(* Schneider Machine Expert - Basic project Control banda, file version 2.9.0.0 *)
(* ProjectInformations: Name=New project *)

HARDWARE
  Cpu 0: TM221CE16R
  EthernetConfiguration: NetworkName=M221, IpAllocationMode=FixedAddress, IpAddress=0.0.0.0, SubnetMask=0.0.0.0
  SerialLineConfiguration: Baud=Baud19200, Parity=ParityEven, DataBits=DataBits8, StopBits=StopBits1, PhysicalMedium=PhysicalMediumRs485, TransmissionMode=TransmissionModeModbusRtu, SlaveId=1, Addressing=SlaveAddressing
  MastTask: UsePeriodScanMode=false, PeriodScan=100
  FastTask: Period=255
  CpuBehavior: StartingMode=StartAsPreviousState, AutoSaveRamOnEeprom=true, WatchdogPeriod=250

SYMBOLS  (address, symbol, comment, settings)
  %M0       AT_EXIT
  %M1       START_FIO
  %M2       RESET_FIO
  %M3       STOP_FIO
  %M4       EMERG_FIO
  %M10      ENTRY_CONVEY
  %M11      STOP_BLAE
  %M12      EXIT_CONVEYOR
  %M13      SORTER_1_TURN
  %M14      SORTER_1_BELT
  %M15      SORTER_2_TURN
  %M16      SORTER_2_BELT
  %M17      SORTER_3_TURN
  %M18      SORTER_3_BELT
  %M19      START_LIGHT
  %M21      STOP_LIGHT
  %M30      START_REMOT
  %M31      STOP_REMOTO
  %M32      PAUSE_REM
  %M33      RESET_REMOT
  %M34      EMERG_REMOTA_
  %M41      BLUE_ACTIVE
  %M42      GREEN_ACTIVE
  %M43      METAL_ACTIVE
  %S6       SB_TB1S  "Time base of 1 s generated by an internal clock"
  %TM0        [Preset=3, Base=OneHundredMilliSeconds]
  %TM1        [Preset=22, Base=OneHundredMilliSeconds]
  %TM2        [Preset=40, Base=OneHundredMilliSeconds]
  %TM10       [Type=TP, Preset=10, Base=OneHundredMilliSeconds]
  %TM11       [Type=TP, Preset=10, Base=OneHundredMilliSeconds]
  %TM12       [Type=TP, Preset=10, Base=OneHundredMilliSeconds]

POU New POU
  (* SectionNumber=1 *)

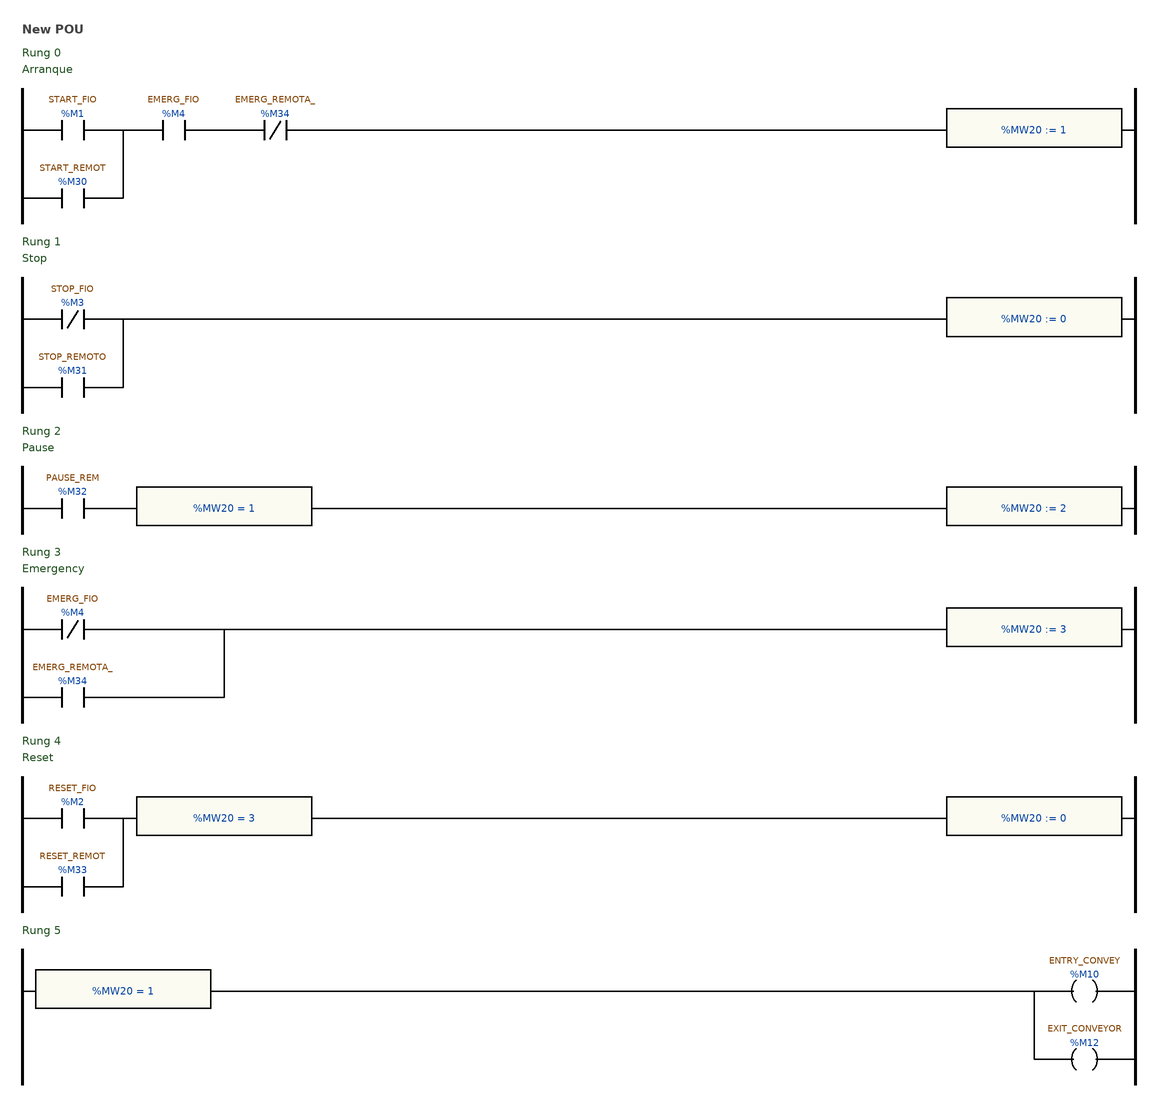

// Rung 0
// Arranque
  LD %M1                  (* START_FIO *)
  OR %M30                 (* START_REMOT *)
  AND %M4                 (* EMERG_FIO *)
  ANDN %M34               (* EMERG_REMOTA_ *)
  [ %MW20 := 1 ]
  // as ST:
  //   IF (START_FIO OR START_REMOT) AND EMERG_FIO AND NOT EMERG_REMOTA_ THEN %MW20 := 1; END_IF;

// Rung 1
// Stop
  LDN %M3                 (* STOP_FIO *)
  OR %M31                 (* STOP_REMOTO *)
  [ %MW20 := 0 ]
  // as ST:
  //   IF NOT STOP_FIO OR STOP_REMOTO THEN %MW20 := 0; END_IF;

// Rung 2
// Pause
  LD %M32                 (* PAUSE_REM *)
  AND [ %MW20 = 1 ]
  [ %MW20 := 2 ]
  // as ST:
  //   IF PAUSE_REM AND %MW20 = 1 THEN %MW20 := 2; END_IF;

// Rung 3
// Emergency
  LDN %M4                 (* EMERG_FIO *)
  OR %M34                 (* EMERG_REMOTA_ *)
  [ %MW20 := 3 ]
  // as ST:
  //   IF NOT EMERG_FIO OR EMERG_REMOTA_ THEN %MW20 := 3; END_IF;

// Rung 4
// Reset
  LD %M2                  (* RESET_FIO *)
  OR %M33                 (* RESET_REMOT *)
  AND [ %MW20 = 3 ]
  [ %MW20 := 0 ]
  // as ST:
  //   IF (RESET_FIO OR RESET_REMOT) AND %MW20 = 3 THEN %MW20 := 0; END_IF;

// Rung 5
  LD [ %MW20 = 1 ]
  ST %M10                 (* ENTRY_CONVEY *)
  ST %M12                 (* EXIT_CONVEYOR *)
  // as ST:
  //   ENTRY_CONVEY := %MW20 = 1;
  //   EXIT_CONVEYOR := %MW20 = 1;

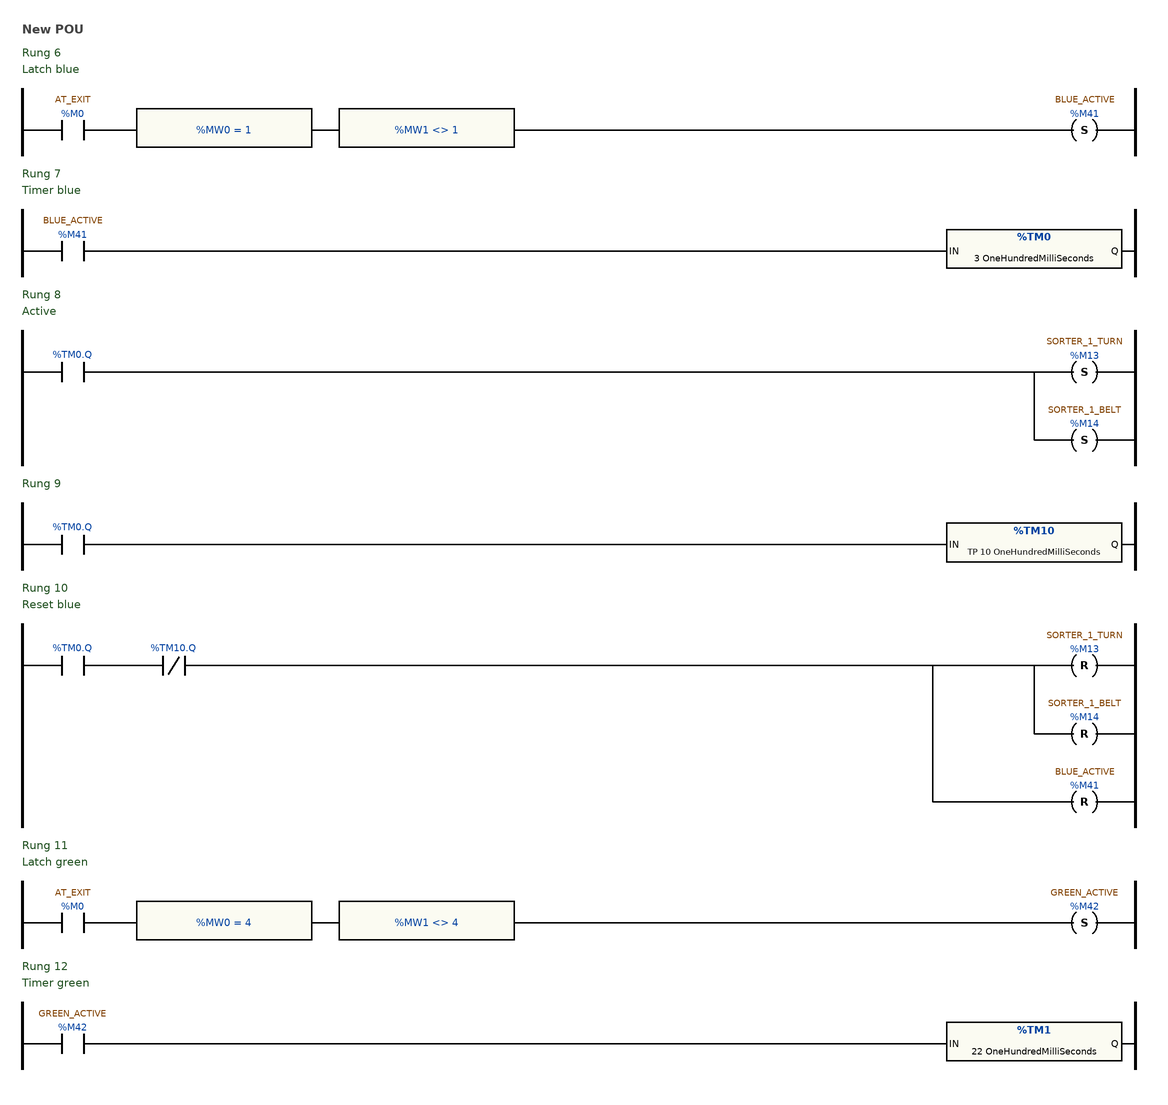

// Rung 6
// Latch blue
  LD %M0                  (* AT_EXIT *)
  AND [ %MW0 = 1 ]
  AND [ %MW1 <> 1 ]
  S %M41                  (* BLUE_ACTIVE *)
  // as ST:
  //   IF AT_EXIT AND %MW0 = 1 AND %MW1 <> 1 THEN BLUE_ACTIVE := TRUE; END_IF;

// Rung 7
// Timer blue
  BLK %TM0
  LD %M41                 (* BLUE_ACTIVE *)
  IN
  END_BLK
  // as ST:
  //   %TM0(IN := BLUE_ACTIVE);

// Rung 8
// Active
  LD %TM0.Q
  S %M13                  (* SORTER_1_TURN *)
  S %M14                  (* SORTER_1_BELT *)
  // as ST:
  //   IF %TM0.Q THEN SORTER_1_TURN := TRUE; END_IF;
  //   IF %TM0.Q THEN SORTER_1_BELT := TRUE; END_IF;

// Rung 9
  BLK %TM10
  LD %TM0.Q
  IN
  END_BLK
  // as ST:
  //   %TM10(IN := %TM0.Q);

// Rung 10
// Reset blue
  LD %TM0.Q
  ANDN %TM10.Q
  R %M13                  (* SORTER_1_TURN *)
  R %M14                  (* SORTER_1_BELT *)
  R %M41                  (* BLUE_ACTIVE *)
  // as ST:
  //   IF %TM0.Q AND NOT %TM10.Q THEN SORTER_1_TURN := FALSE; END_IF;
  //   IF %TM0.Q AND NOT %TM10.Q THEN SORTER_1_BELT := FALSE; END_IF;
  //   IF %TM0.Q AND NOT %TM10.Q THEN BLUE_ACTIVE := FALSE; END_IF;

// Rung 11
// Latch green
  LD %M0                  (* AT_EXIT *)
  AND [ %MW0 = 4 ]
  AND [ %MW1 <> 4 ]
  S %M42                  (* GREEN_ACTIVE *)
  // as ST:
  //   IF AT_EXIT AND %MW0 = 4 AND %MW1 <> 4 THEN GREEN_ACTIVE := TRUE; END_IF;

// Rung 12
// Timer green
  BLK %TM1
  LD %M42                 (* GREEN_ACTIVE *)
  IN
  END_BLK
  // as ST:
  //   %TM1(IN := GREEN_ACTIVE);

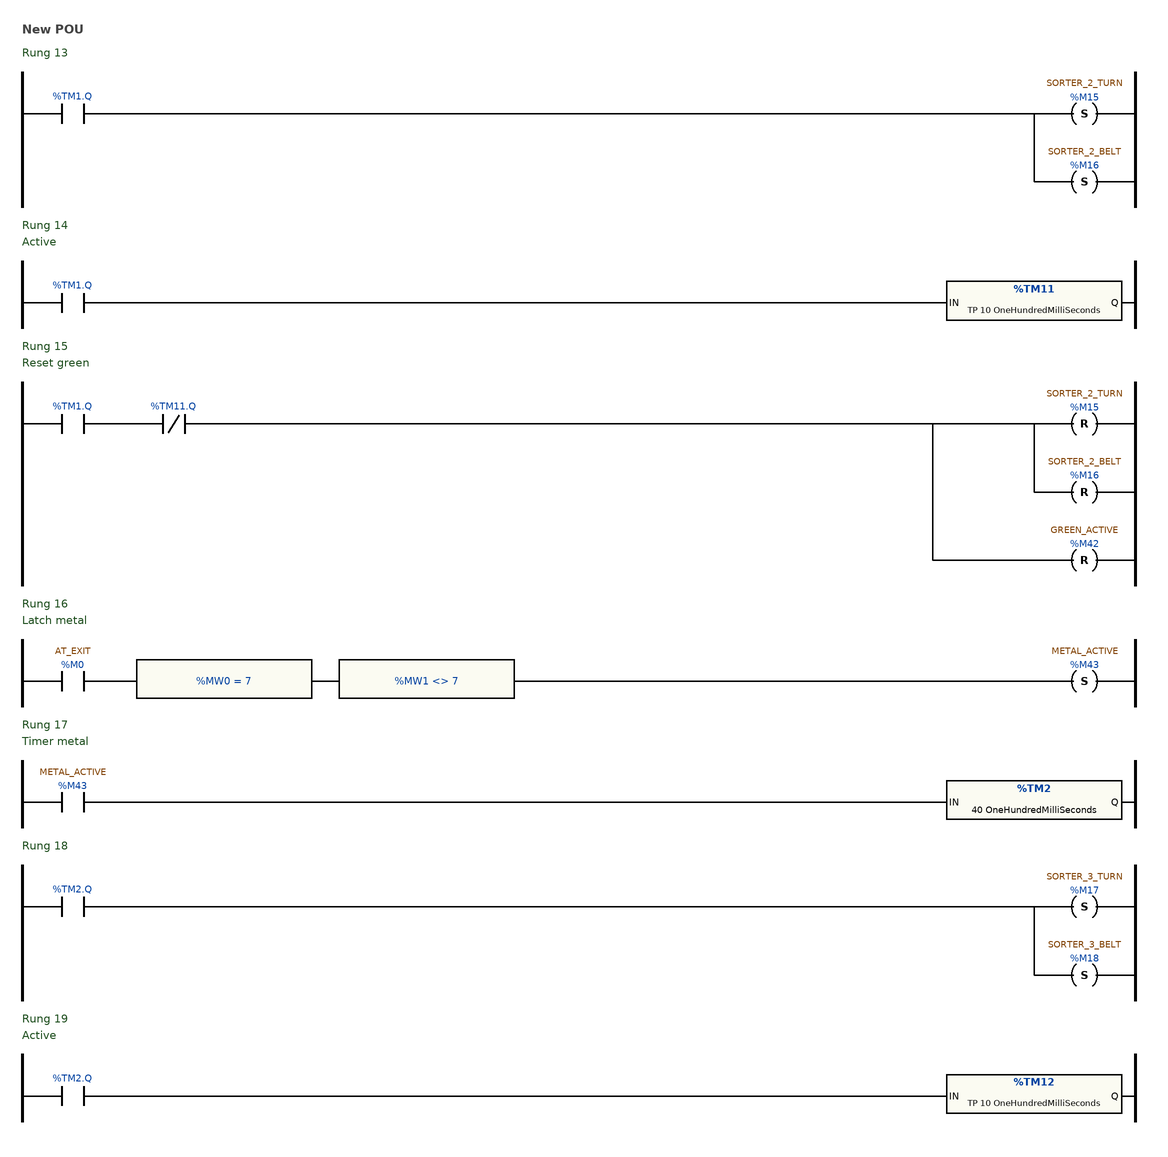

// Rung 13
  LD %TM1.Q
  S %M15                  (* SORTER_2_TURN *)
  S %M16                  (* SORTER_2_BELT *)
  // as ST:
  //   IF %TM1.Q THEN SORTER_2_TURN := TRUE; END_IF;
  //   IF %TM1.Q THEN SORTER_2_BELT := TRUE; END_IF;

// Rung 14
// Active
  BLK %TM11
  LD %TM1.Q
  IN
  END_BLK
  // as ST:
  //   %TM11(IN := %TM1.Q);

// Rung 15
// Reset green
  LD %TM1.Q
  ANDN %TM11.Q
  R %M15                  (* SORTER_2_TURN *)
  R %M16                  (* SORTER_2_BELT *)
  R %M42                  (* GREEN_ACTIVE *)
  // as ST:
  //   IF %TM1.Q AND NOT %TM11.Q THEN SORTER_2_TURN := FALSE; END_IF;
  //   IF %TM1.Q AND NOT %TM11.Q THEN SORTER_2_BELT := FALSE; END_IF;
  //   IF %TM1.Q AND NOT %TM11.Q THEN GREEN_ACTIVE := FALSE; END_IF;

// Rung 16
// Latch metal
  LD %M0                  (* AT_EXIT *)
  AND [ %MW0 = 7 ]
  AND [ %MW1 <> 7 ]
  S %M43                  (* METAL_ACTIVE *)
  // as ST:
  //   IF AT_EXIT AND %MW0 = 7 AND %MW1 <> 7 THEN METAL_ACTIVE := TRUE; END_IF;

// Rung 17
// Timer metal
  BLK %TM2
  LD %M43                 (* METAL_ACTIVE *)
  IN
  END_BLK
  // as ST:
  //   %TM2(IN := METAL_ACTIVE);

// Rung 18
  LD %TM2.Q
  S %M17                  (* SORTER_3_TURN *)
  S %M18                  (* SORTER_3_BELT *)
  // as ST:
  //   IF %TM2.Q THEN SORTER_3_TURN := TRUE; END_IF;
  //   IF %TM2.Q THEN SORTER_3_BELT := TRUE; END_IF;

// Rung 19
// Active
  BLK %TM12
  LD %TM2.Q
  IN
  END_BLK
  // as ST:
  //   %TM12(IN := %TM2.Q);

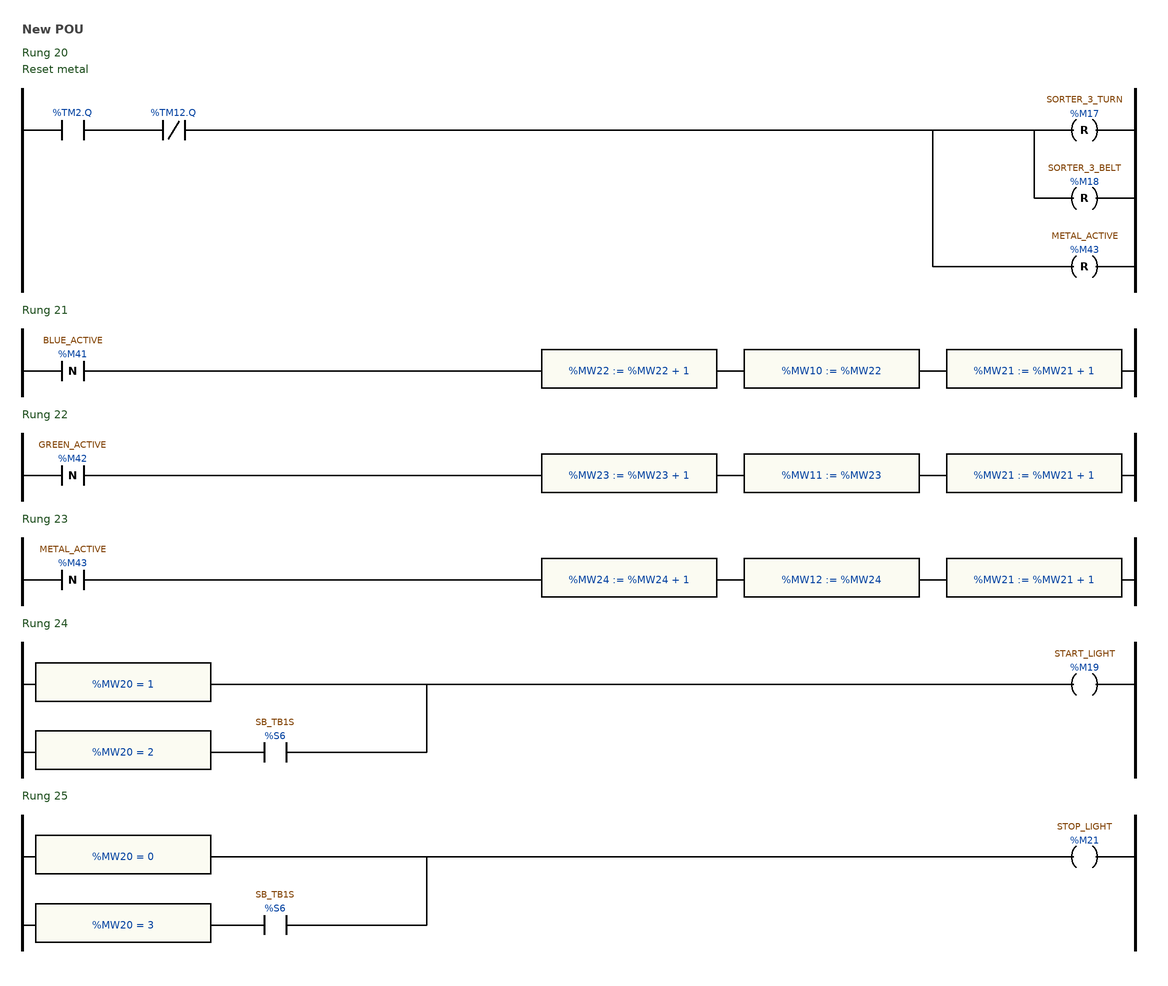

// Rung 20
// Reset metal
  LD %TM2.Q
  ANDN %TM12.Q
  R %M17                  (* SORTER_3_TURN *)
  R %M18                  (* SORTER_3_BELT *)
  R %M43                  (* METAL_ACTIVE *)
  // as ST:
  //   IF %TM2.Q AND NOT %TM12.Q THEN SORTER_3_TURN := FALSE; END_IF;
  //   IF %TM2.Q AND NOT %TM12.Q THEN SORTER_3_BELT := FALSE; END_IF;
  //   IF %TM2.Q AND NOT %TM12.Q THEN METAL_ACTIVE := FALSE; END_IF;

// Rung 21
  LDF %M41                (* BLUE_ACTIVE *)
  OPER [ %MW22 := %MW22 + 1 ]
  OPER [ %MW10 := %MW22 ]
  [ %MW21 := %MW21 + 1 ]
  // as ST:
  //   IF FALLING(BLUE_ACTIVE) THEN %MW22 := %MW22 + 1; END_IF;
  //   IF FALLING(BLUE_ACTIVE) THEN %MW10 := %MW22; END_IF;
  //   IF FALLING(BLUE_ACTIVE) THEN %MW21 := %MW21 + 1; END_IF;

// Rung 22
  LDF %M42                (* GREEN_ACTIVE *)
  OPER [ %MW23 := %MW23 + 1 ]
  OPER [ %MW11 := %MW23 ]
  [ %MW21 := %MW21 + 1 ]
  // as ST:
  //   IF FALLING(GREEN_ACTIVE) THEN %MW23 := %MW23 + 1; END_IF;
  //   IF FALLING(GREEN_ACTIVE) THEN %MW11 := %MW23; END_IF;
  //   IF FALLING(GREEN_ACTIVE) THEN %MW21 := %MW21 + 1; END_IF;

// Rung 23
  LDF %M43                (* METAL_ACTIVE *)
  OPER [ %MW24 := %MW24 + 1 ]
  OPER [ %MW12 := %MW24 ]
  [ %MW21 := %MW21 + 1 ]
  // as ST:
  //   IF FALLING(METAL_ACTIVE) THEN %MW24 := %MW24 + 1; END_IF;
  //   IF FALLING(METAL_ACTIVE) THEN %MW12 := %MW24; END_IF;
  //   IF FALLING(METAL_ACTIVE) THEN %MW21 := %MW21 + 1; END_IF;

// Rung 24
  LD [ %MW20 = 1 ]
  OR( [ %MW20 = 2 ]
  AND %S6                 (* SB_TB1S *)
  )
  ST %M19                 (* START_LIGHT *)
  // as ST:
  //   START_LIGHT := %MW20 = 1 OR %MW20 = 2 AND SB_TB1S;

// Rung 25
  LD [ %MW20 = 0 ]
  OR( [ %MW20 = 3 ]
  AND %S6                 (* SB_TB1S *)
  )
  ST %M21                 (* STOP_LIGHT *)
  // as ST:
  //   STOP_LIGHT := %MW20 = 0 OR %MW20 = 3 AND SB_TB1S;
